// TIA Portal V16 export
// export: Created 2021-08-10T09:04:59.3532102Z, ExportSetting WithDefaults, WithReadOnly, DisplayName Totally Integrated Automation Portal, DisplayVersion V16, DisplayName TIA Portal Version Control Interface, DisplayVersion V16, DisplayName TIA Portal Openness, DisplayVersion V16, DisplayName TIA Portal Teamcenter Gateway, DisplayVersion V16, DisplayName SINAMICS Startdrive Advanced, DisplayVersion V16, DisplayName SINAMICS Startdrive G130, G150, S120, S150, SINAMICS MV, S210, DisplayVersion V16, DisplayName SINAMICS Startdrive G110M, G120, G120C, G120D, G120P, DisplayVersion V16, DisplayName STEP 7 Professional, DisplayVersion V16, DisplayName STEP 7 Safety, DisplayVersion V16, DisplayName WinCC Unified SCADA Engineering System, DisplayVersion V16
ORGANIZATION_BLOCK "Main"   // OB1, FBD, ProgramCycle
TITLE = "Main Program Sweep (Cycle)"
{ S7_Optimized_Access := 'TRUE' }
VERSION : 0.1
// stored: AutoNumber true, CodeModifiedDate 2021-08-10T08:54:10.1985647Z, CompileDate 2021-08-10T08:57:18.4266346Z, ConstantName OB_Main, CreationDate 2020-02-26T07:01:34.5488912Z, EventClass Program cycle, HandleErrorsWithinBlock false, InterfaceModifiedDate 2008-07-21T16:55:08.419547Z, IsConsistent true, IsIECCheckEnabled false, IsKnowHowProtected false, IsWriteProtected false, ModifiedDate 2021-08-10T08:54:10.1985647Z, ParameterModified 2008-07-21T16:55:08.419547Z, PLCSimAdvancedSupport true, PriorityNumber 1, ProcessImagePartNumber 65535, SetENOAutomatically false, StructureModified 2008-07-21T16:55:08.419547Z
   VAR_INPUT
      Initial_Call : Bool;   // Initial call of this OB
      Remanence : Bool;   // =True, if remanent data are available
   END_VAR
BEGIN

REGION Network 1
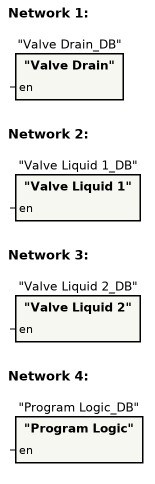
   "Valve Drain_DB"();   // "Valve Drain"
END_REGION

REGION Network 2
   "Valve Liquid 1_DB"();   // "Valve Liquid 1"
END_REGION

REGION Network 3
   "Valve Liquid 2_DB"();   // "Valve Liquid 2"
END_REGION

REGION Network 4
   "Program Logic_DB"();   // "Program Logic"
END_REGION
END_ORGANIZATION_BLOCK
